PROGRAM MAIN
VAR
END_VAR

END_PROGRAM

(* stored: Version 1.1.0.1
   POU MAIN: Id {62af5e7f-d16b-4657-b275-2b4eba6f9baa} *)
